(* PLC project Tc2_Utilities.ULARGE_INTEGER Demo, tc3-libraries-kb TwinCAT 3.1 *)
(* stored: creationDateTime 2026-05-10T18:00:00, modificationDateTime 2026-05-10T18:00:00 *)

PROGRAM P_Demo_ULARGE_INTEGER
  VAR
    rResult : T_ULARGE_INTEGER;  (* ULARGE_INTEGER 返回值 *)
    bRun : BOOL;  (* 触发一次调用 *)
    result : T_ULARGE_INTEGER;  (* 测试用本地变量 *)
  END_VAR

            // ============================================================
// Tc2_Utilities.ULARGE_INTEGER 演示程序（FUNCTION）
// ============================================================
// 验证步骤：
//   1. 引用 Tc2_Utilities
//   2. 编译 + 登录
//   3. 强制 bRun := TRUE 一个周期
//   4. 在线监视 rResult
// ============================================================

IF bRun THEN
    rResult := ULARGE_INTEGER(0, 16#12345678);
    bRun := FALSE;
END_IF;

          
END_PROGRAM
